(* PLC project waste_water_treatment_facility, Generated TextualNotationConverter 1.0 *)
(* stored: creationDateTime 2025-07-30T12:00:00, modificationDateTime 2025-01-30T12:00:00 *)

FUNCTION_BLOCK ANALOG_IN
  VAR_INPUT
    Name : STRING;
    Description : STRING;
    Raw_Signal : REAL;
    PV_High : REAL;
    PV_Low : REAL;
    Scaling_Slope : REAL;
    Scaling_Offset : REAL;
    Alarm_Enable : BOOL;
  END_VAR
  VAR_OUTPUT
    PV : REAL;
    High_Alarm : BOOL;
    Low_Alarm : BOOL;
    General_Fault : BOOL;
  END_VAR

            
          
END_FUNCTION_BLOCK

FUNCTION_BLOCK MOTOR_VSD
  VAR_INPUT
    Name : STRING;
    Description : STRING;
    Start_Cmd : BOOL;
    Stop_Cmd : BOOL;
    Speed_SP : REAL;
    Accel_Ramp : STRING;
    Decel_Ramp : STRING;
    Inhibit : BOOL;
  END_VAR
  VAR_OUTPUT
    Speed_Out : REAL;
    FB_Running : BOOL;
    FB_Fault : BOOL;
    FB_Ready : BOOL;
    FB_ActualSpeed : REAL;
    Alarm_Speed_Deviation : BOOL;
    Alarm_Comm_Fail : BOOL;
  END_VAR

            
          
END_FUNCTION_BLOCK

FUNCTION_BLOCK PID_BASIC
  VAR_INPUT
    Name : STRING;
    Description : STRING;
    AUTO : BOOL;
    PV : REAL;
    SP : REAL;
    MV_MIN : REAL;
    MV_MAX : REAL;
    X0 : REAL;
    KP : REAL;
    TR : REAL;
    TD : REAL;
    PV_High : REAL;
    PV_Low : REAL;
    Deviation_Limit : REAL;
    Inhibit : BOOL;
  END_VAR
  VAR_OUTPUT
    PV_High_Alarm : BOOL;
    PV_Low_Alarm : BOOL;
    Deviation_Alarm : BOOL;
    XOUT : REAL;
  END_VAR

            
          
END_FUNCTION_BLOCK

PROGRAM Section5
  VAR
    PH_401_pH_PV : REAL;
    AC_401_Alkalinity_PV : REAL;
    FT_101_InfluentFlow_PV : REAL;
    LT_401_TankLevel_PV : REAL;
    TS_401_Temperature_PV : REAL;
    PIC_401_pH_MV_Percent : REAL;
    PIC_402_Alkalinity_MV_Percent : REAL;
  END_VAR
  VAR
    AC-401 : ANALOG_IN;
    CD-401 : MOTOR_VSD;
    FT-101 : ANALOG_IN;
    LT-401 : ANALOG_IN;
    PH-401 : ANALOG_IN;
    PIC-401 : PID_BASIC;
    PIC-402 : PID_BASIC;
    TS-401 : ANALOG_IN;
  END_VAR
  VAR  (* added by the conversion: wires and edge detectors of the diagram *)
    _OR3_OUT : BOOL;
  END_VAR

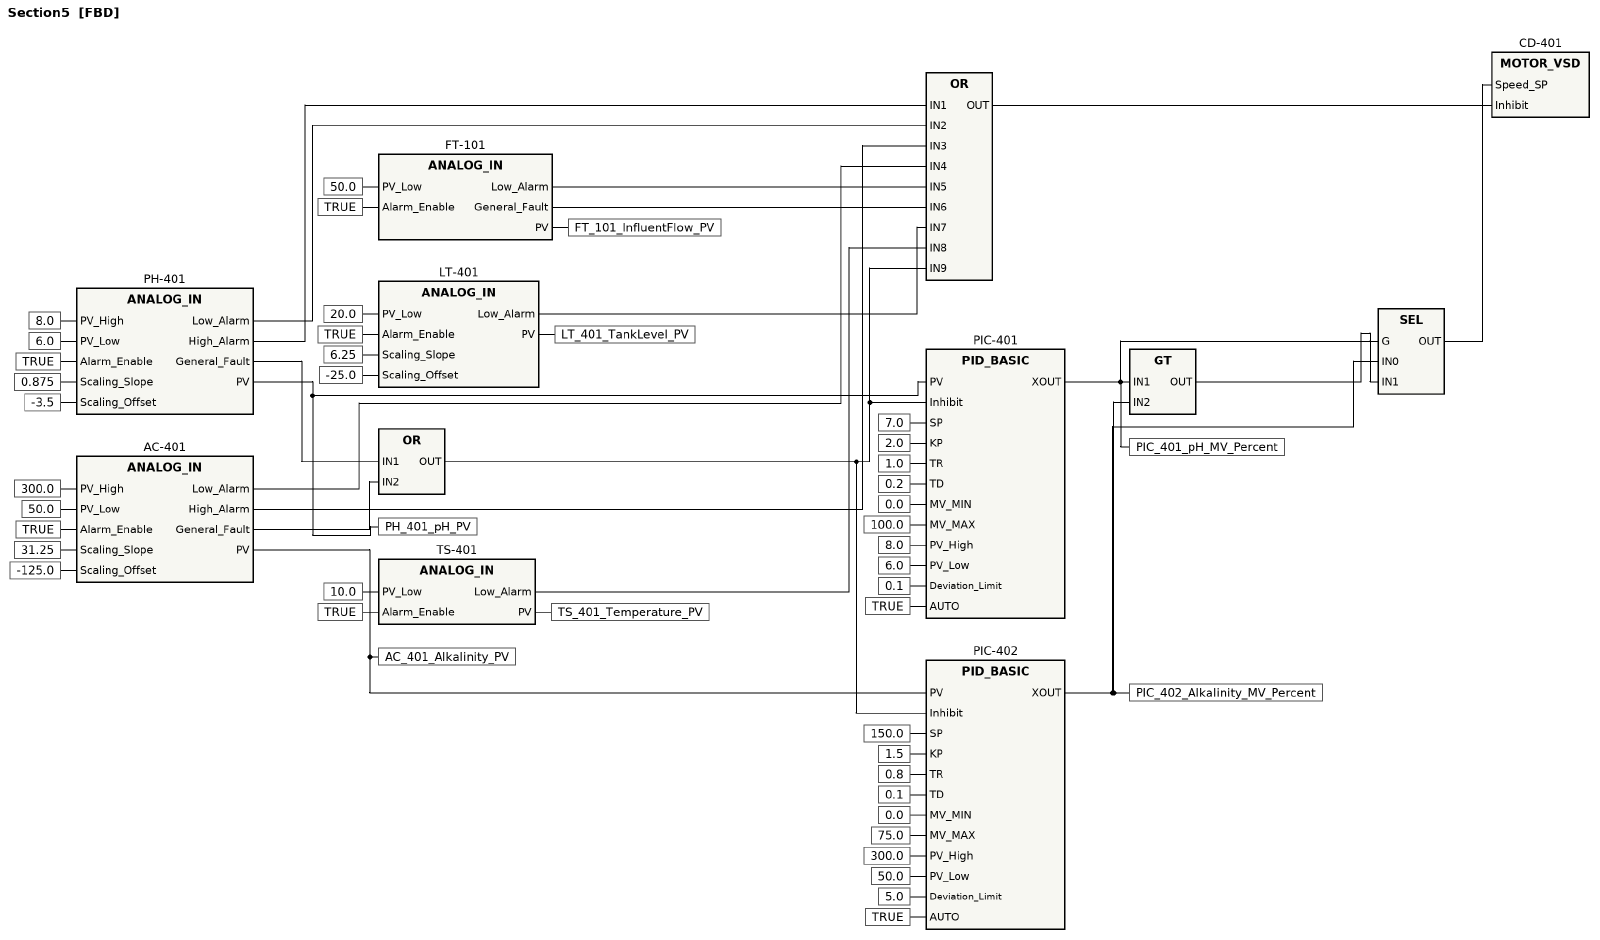
(* FBD diagram, written out as Structured Text *)
AC-401(PV_High := 300.0, PV_Low := 50.0, Alarm_Enable := TRUE, Scaling_Slope := 31.25, Scaling_Offset := -125.0);
AC_401_Alkalinity_PV := AC-401.PV;
FT-101(PV_Low := 50.0, Alarm_Enable := TRUE);
FT_101_InfluentFlow_PV := FT-101.PV;
LT-401(PV_Low := 20.0, Alarm_Enable := TRUE, Scaling_Slope := 6.25, Scaling_Offset := -25.0);
LT_401_TankLevel_PV := LT-401.PV;
PH-401(PV_High := 8.0, PV_Low := 6.0, Alarm_Enable := TRUE, Scaling_Slope := 0.875, Scaling_Offset := -3.5);
PH_401_pH_PV := PH-401.PV;
_OR3_OUT := PH-401.General_Fault OR AC-401.General_Fault;
PIC-401(PV := PH-401.PV, Inhibit := _OR3_OUT, SP := 7.0, KP := 2.0, TR := 1.0, TD := 0.2, MV_MIN := 0.0, MV_MAX := 100.0, PV_High := 8.0, PV_Low := 6.0, Deviation_Limit := 0.1, AUTO := TRUE);
PIC_401_pH_MV_Percent := PIC-401.XOUT;
PIC-402(PV := AC-401.PV, Inhibit := _OR3_OUT, SP := 150.0, KP := 1.5, TR := 0.8, TD := 0.1, MV_MIN := 0.0, MV_MAX := 75.0, PV_High := 300.0, PV_Low := 50.0, Deviation_Limit := 5.0, AUTO := TRUE);
PIC_402_Alkalinity_MV_Percent := PIC-402.XOUT;
TS-401(PV_Low := 10.0, Alarm_Enable := TRUE);
TS_401_Temperature_PV := TS-401.PV;
CD-401(Speed_SP := SEL(PIC-401.XOUT > PIC-402.XOUT, PIC-402.XOUT, PIC-401.XOUT), Inhibit := PH-401.High_Alarm OR PH-401.Low_Alarm OR AC-401.High_Alarm OR AC-401.Low_Alarm OR FT-101.Low_Alarm OR FT-101.General_Fault OR LT-401.Low_Alarm OR TS-401.Low_Alarm OR _OR3_OUT);
END_PROGRAM

FUNCTION_BLOCK BOOL_IN
  VAR_INPUT
    Name : STRING;
    Description : STRING;
    Bool_In : BOOL;
    Alarm_OnTrue : BOOL;
    Alarm_OnFalse : BOOL;
    Latch_Enable : BOOL;
    Reset_Latch : BOOL;
  END_VAR
  VAR_OUTPUT
    Bool_Out : BOOL;
    Alarm_Active : BOOL;
    Latched_Status : BOOL;
  END_VAR

            
          
END_FUNCTION_BLOCK

FUNCTION_BLOCK DIGITAL_IN
  VAR_INPUT
    Name : STRING;
    Description : STRING;
    DI_Raw : BOOL;
    DebounceTime : STRING;
    EnableAlarm : BOOL;
  END_VAR
  VAR_OUTPUT
    DI_Out : BOOL;
    Fault_State : BOOL;
  END_VAR

            
          
END_FUNCTION_BLOCK

FUNCTION_BLOCK DUTY_STANDBY
  VAR_INPUT
    Name : STRING;
    Description : STRING;
    Enable : BOOL;
    StartRequest : BOOL;
    AlternateEnable : BOOL;
    ForcePumpA : BOOL;
    ForcePumpB : BOOL;
    DutyElapsed : BOOL;
    MinRunElapsed : BOOL;
    SwitchoverDelayElapsed : BOOL;
    StartTimeoutElapsed : BOOL;
    PumpA_RunFB : BOOL;
    PumpB_RunFB : BOOL;
    PumpA_Fault : BOOL;
    PumpB_Fault : BOOL;
    Reset : BOOL;
    Inhibit : BOOL;
  END_VAR
  VAR_OUTPUT
    CmdPumpA : BOOL;
    CmdPumpB : BOOL;
    ActiveIsA : BOOL;
    SwitchedDueToDuty : BOOL;
    SwitchedDueToFailure : BOOL;
    Alarm_FailedStart_A : BOOL;
    Alarm_FailedStart_B : BOOL;
    Alarm_NoAvailablePump : BOOL;
  END_VAR

            
          
END_FUNCTION_BLOCK

FUNCTION_BLOCK MOTOR_2SPD
  VAR_INPUT
    Name : STRING;
    Description : STRING;
    Start_Cmd : BOOL;
    Stop_Cmd : BOOL;
    Speed_High_Cmd : BOOL;
    Speed_Low_Cmd : BOOL;
    Inhibit : BOOL;
  END_VAR
  VAR_OUTPUT
    Motor_Start_Out : BOOL;
    FB_Running : BOOL;
    FB_Trip : BOOL;
    FB_HighSpeed : BOOL;
    FB_LowSpeed : BOOL;
    Alarm_Speed_Error : BOOL;
  END_VAR

            
          
END_FUNCTION_BLOCK

FUNCTION_BLOCK MOTOR_ON_OFF
  VAR_INPUT
    Name : STRING;
    Description : STRING;
    Start_Cmd : BOOL;
    Stop_Cmd : BOOL;
    Start_Delay : STRING;
    MinRunTime : STRING;
    Inhibit : BOOL;
  END_VAR
  VAR_OUTPUT
    Motor_Start_Out : BOOL;
    FB_Running : BOOL;
    FB_Trip : BOOL;
    Alarm_Start_Fail : BOOL;
    Alarm_Stop_Fail : BOOL;
  END_VAR

            
          
END_FUNCTION_BLOCK

FUNCTION_BLOCK RATIO_CONTROL
  VAR_INPUT
    Name : STRING;
    Description : STRING;
    Auto : BOOL;
    PrimaryPV : REAL;
    SecondaryPV : REAL;
    RatioSP : REAL;
    Bias : REAL;
    TrimKp : REAL;
    TrimTi : STRING;
    MV_MIN : REAL;
    MV_MAX : REAL;
    ManOut : REAL;
    Inhibit : BOOL;
  END_VAR
  VAR_OUTPUT
    SlaveSP : REAL;
    ActiveRatio : REAL;
    RatioErr : REAL;
  END_VAR

            
          
END_FUNCTION_BLOCK

FUNCTION_BLOCK SPLIT_RANGE
  VAR_INPUT
    Name : STRING;
    Description : STRING;
    IN : REAL;
    Split_Point : REAL;
    Output1_Start : REAL;
    Output1_End : REAL;
    Output2_Start : REAL;
    Output2_End : REAL;
  END_VAR
  VAR_OUTPUT
    OUT1 : REAL;
    OUT2 : REAL;
  END_VAR

            
          
END_FUNCTION_BLOCK

FUNCTION_BLOCK VALVE_ELECTRIC
  VAR_INPUT
    Name : STRING;
    Description : STRING;
    Control_Signal : REAL;
    Manual_Mode : BOOL;
    Manual_Position : REAL;
    Open_Limit : REAL;
    Close_Limit : REAL;
    Timeout : STRING;
    Inhibit : BOOL;
  END_VAR
  VAR_OUTPUT
    Valve_Position : REAL;
    Feedback_Pos : REAL;
    Valve_Moving : BOOL;
    Position_Error : BOOL;
    Alarm : BOOL;
  END_VAR

            
          
END_FUNCTION_BLOCK

FUNCTION_BLOCK VALVE_ON_OFF
  VAR_INPUT
    Name : STRING;
    Description : STRING;
    Open_Cmd : BOOL;
    Close_Cmd : BOOL;
    Timeout : STRING;
    Inhibit : BOOL;
  END_VAR
  VAR_OUTPUT
    FB_Opened : BOOL;
    FB_Closed : BOOL;
    Valve_Open_Out : BOOL;
    Valve_Close_Out : BOOL;
    Alarm_Position_Error : BOOL;
    Alarm_General : BOOL;
  END_VAR

            
          
END_FUNCTION_BLOCK

FUNCTION_BLOCK VOTING_ANALOG
  VAR_INPUT
    Name : STRING;
    Description : STRING;
    Input1 : REAL;
    Input2 : REAL;
    Input3 : REAL;
    Deviation_Limit : REAL;
    Voting_Scheme : STRING;
    EnableAlarm : BOOL;
    Inhibit : BOOL;
  END_VAR
  VAR_OUTPUT
    Voted_Output : REAL;
    Sensor1_Fault : BOOL;
    Sensor2_Fault : BOOL;
    Sensor3_Fault : BOOL;
    Alarm_Voting_Error : BOOL;
    Healthy_Sensors_Count : INT;
  END_VAR

            
          
END_FUNCTION_BLOCK

PROGRAM Section6
  VAR
    FFIC-102_AirflowSP_for_FIC-103 : REAL;
    PT-501_AirHeaderPressure_PV : REAL;
    B-501A_Running_FB : BOOL;
    B-501B_Running_FB : BOOL;
    MX-501_Running_FB : BOOL;
    XV-105_Open_FB : BOOL;
    AirflowDeviationAlarm : BOOL;
    LowFlowAlarm : BOOL;
  END_VAR
  VAR
    B-501A : MOTOR_ON_OFF;
    B-501B : MOTOR_ON_OFF;
    FFIC-102 : RATIO_CONTROL;
    FIC-101 : PID_BASIC;
    FIC-103 : PID_BASIC;
    FV-102 : VALVE_ELECTRIC;
    MX-501 : MOTOR_ON_OFF;
    PT-501 : ANALOG_IN;
    XV-105 : VALVE_ON_OFF;
  END_VAR
  VAR  (* added by the conversion: wires and edge detectors of the diagram *)
    _OR61_IN4 : ANY;
    _OR61_IN3 : ANY;
    _OR61_IN5 : ANY;
    _OR61_IN6 : ANY;
    _OR61_IN1 : ANY;
    _OR61_IN2 : ANY;
    _OR61_OUT : ANY;
    _OR61_OUT_2 : BOOL;
    _OR63_IN2 : ANY;
    _OR63_OUT : ANY;
    _OR63_OUT_2 : BOOL;
    _OR58_IN2 : ANY;
    _OR58_OUT : BOOL;
  END_VAR

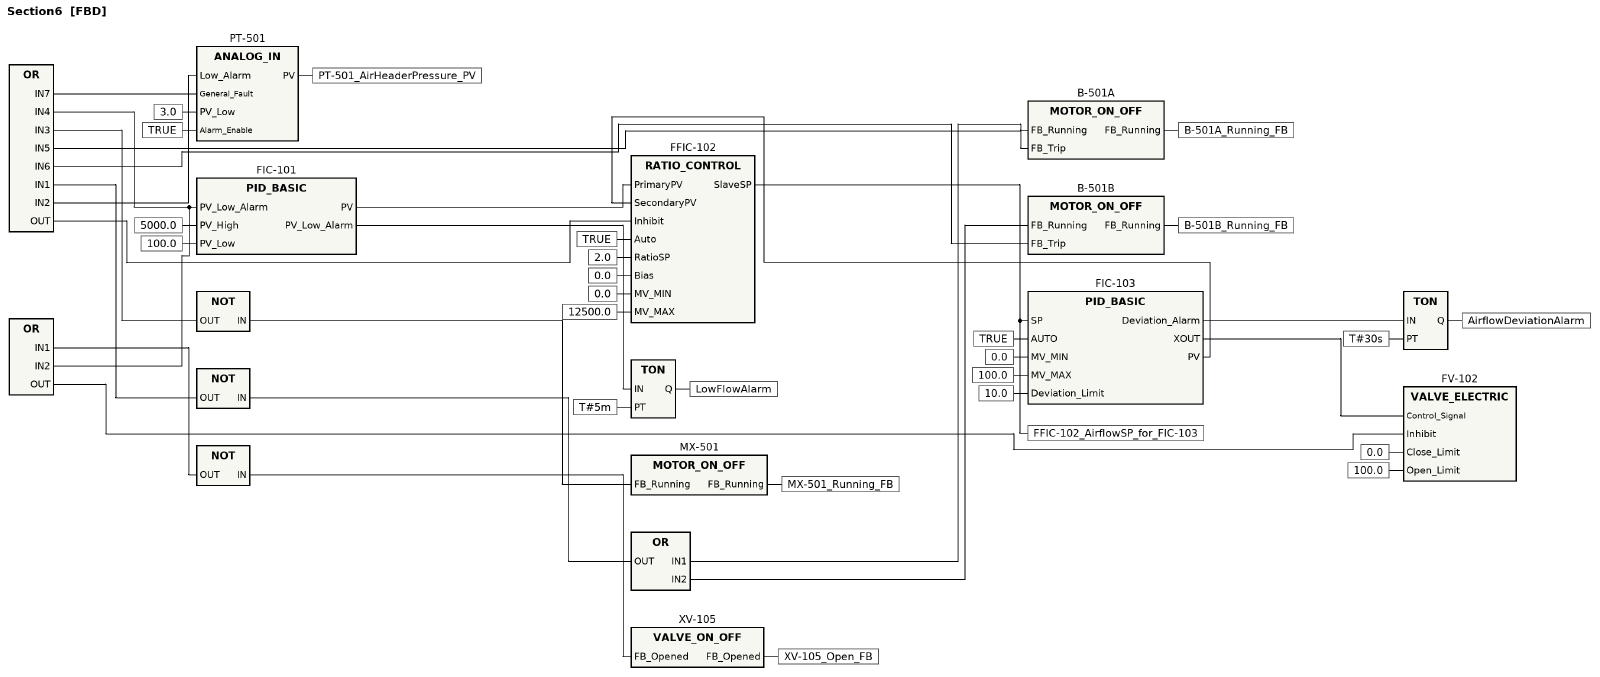
(* FBD diagram, written out as Structured Text *)
_OR61_OUT_2 := OR(IN4 => _OR61_IN4, IN3 => _OR61_IN3, IN5 => _OR61_IN5, IN6 => _OR61_IN6, IN1 => _OR61_IN1, IN2 => _OR61_IN2, OUT => _OR61_OUT);
_OR63_OUT_2 := OR(IN2 => _OR63_IN2, OUT => _OR63_OUT);
FIC-101(PV_Low_Alarm := _OR61_IN4 OR _OR63_IN2, PV_High := 5000.0, PV_Low := 100.0);
FFIC-102(PrimaryPV := FIC-101.PV, SecondaryPV := FIC-103.PV, Inhibit := _OR61_OUT, Auto := TRUE, RatioSP := 2.0, Bias := 0.0, MV_MIN := 0.0, MV_MAX := 12500.0);
FIC-103(SP := FFIC-102.SlaveSP, AUTO := TRUE, MV_MIN := 0.0, MV_MAX := 100.0, Deviation_Limit := 10.0);
AirflowDeviationAlarm := TON(FIC-103.Deviation_Alarm, T#30s);
_OR58_OUT := OR(OUT := NOT _OR61_IN1, IN2 => _OR58_IN2);
B-501A(FB_Running := _OR58_OUT, FB_Trip := _OR61_IN5);
B-501A_Running_FB := B-501A.FB_Running;
B-501B(FB_Running := _OR58_IN2, FB_Trip := _OR61_IN6);
B-501B_Running_FB := B-501B.FB_Running;
FFIC-102_AirflowSP_for_FIC-103 := FFIC-102.SlaveSP;
LowFlowAlarm := TON(FIC-101.PV_Low_Alarm, T#5m);
MX-501(FB_Running := NOT _OR61_IN3);
MX-501_Running_FB := MX-501.FB_Running;
PT-501(Low_Alarm := _OR61_IN2, General_Fault := _OR61_OUT_2, PV_Low := 3.0, Alarm_Enable := TRUE);
PT-501_AirHeaderPressure_PV := PT-501.PV;
XV-105(FB_Opened := NOT _OR63_OUT_2);
XV-105_Open_FB := XV-105.FB_Opened;
FV-102(Control_Signal := FIC-103.XOUT, Inhibit := _OR63_OUT, Close_Limit := 0.0, Open_Limit := 100.0);
END_PROGRAM

PROGRAM Section7
  VAR
    PT_601A_DischargePressure_PV : REAL;
    PT_601B_DischargePressure_PV : REAL;
    LS_601_BlanketLevelSwitchStatus : BOOL;
    CL_601A_Running : BOOL;
    CL_601B_Running : BOOL;
    PS_601A_Running : BOOL;
    PS_601B_Running : BOOL;
    VS_601A_Feedback_Position_Pct : REAL;
    VS_601B_Feedback_Position_Pct : REAL;
    CL_601_ActiveIsA : BOOL;
    PS_601_ActiveIsA : BOOL;
    CL_601A_RunCmd : BOOL;
    CL_601B_RunCmd : BOOL;
    PS_601A_RunCmd : BOOL;
    PS_601B_RunCmd : BOOL;
  END_VAR
  VAR
    LS-601 : BOOL_IN;
    PT-601A : ANALOG_IN;
    PT-601B : ANALOG_IN;
    CL-601A : MOTOR_ON_OFF;
    CL-601B : MOTOR_ON_OFF;
    PS-601A : MOTOR_ON_OFF;
    PS-601B : MOTOR_ON_OFF;
    VS-601A : VALVE_ELECTRIC;
    VS-601B : VALVE_ELECTRIC;
    CL-601_DUTY_STANDBY : DUTY_STANDBY;
    PS-601_DUTY_STANDBY : DUTY_STANDBY;
  END_VAR
  VAR  (* added by the conversion: wires and edge detectors of the diagram *)
    _OR110_OUT : BOOL;
    _OR113_OUT : BOOL;
    _OR114_OUT : BOOL;
    _OR100_OUT : BOOL;
    _OR115_OUT : BOOL;
    _OR105_OUT : BOOL;
  END_VAR

(* FBD diagram, written out as Structured Text *)
LS-601(Alarm_OnTrue := TRUE, Alarm_OnFalse := FALSE, Latch_Enable := TRUE);
_OR110_OUT := LS-601.Bool_Out OR LS-601.Alarm_Active;
_OR113_OUT := _OR110_OUT OR CL-601A.FB_Trip;
CL-601A(Start_Cmd := CL-601_DUTY_STANDBY.CmdPumpA, Inhibit := _OR113_OUT, Start_Delay := T#5S, MinRunTime := T#30M);
_OR114_OUT := _OR110_OUT OR CL-601B.FB_Trip;
CL-601B(Start_Cmd := CL-601_DUTY_STANDBY.CmdPumpB, Inhibit := _OR114_OUT, Start_Delay := T#5S, MinRunTime := T#30M);
_OR100_OUT := CL-601A.FB_Running OR CL-601B.FB_Running;
PT-601A(PV_Low := 25.0, Alarm_Enable := TRUE);
PT-601B(PV_Low := 25.0, Alarm_Enable := TRUE);
_OR115_OUT := _OR110_OUT OR PT-601A.Low_Alarm OR PT-601B.Low_Alarm;
CL-601_DUTY_STANDBY(DutyElapsed := TON(_OR100_OUT, T#72H), MinRunElapsed := TON(_OR100_OUT, T#30M), SwitchoverDelayElapsed := TON(NOT _OR100_OUT, T#10S), PumpA_RunFB := CL-601A.FB_Running, PumpB_RunFB := CL-601B.FB_Running, PumpA_Fault := _OR113_OUT, PumpB_Fault := _OR114_OUT, Inhibit := _OR115_OUT, Enable := TRUE, StartRequest := TRUE, AlternateEnable := TRUE);
CL_601A_RunCmd := CL-601_DUTY_STANDBY.CmdPumpA;
CL_601A_Running := CL-601A.FB_Running;
CL_601B_RunCmd := CL-601_DUTY_STANDBY.CmdPumpB;
CL_601B_Running := CL-601B.FB_Running;
CL_601_ActiveIsA := CL-601_DUTY_STANDBY.ActiveIsA;
LS_601_BlanketLevelSwitchStatus := LS-601.Bool_Out;
PS-601A(Start_Cmd := PS-601_DUTY_STANDBY.CmdPumpA, Inhibit := PT-601A.Low_Alarm OR _OR110_OUT, Start_Delay := T#5S, MinRunTime := T#30M);
PS-601B(Start_Cmd := PS-601_DUTY_STANDBY.CmdPumpB, Inhibit := PT-601B.Low_Alarm OR _OR110_OUT, Start_Delay := T#5S, MinRunTime := T#30M);
_OR105_OUT := PS-601A.FB_Running OR PS-601B.FB_Running;
PS-601_DUTY_STANDBY(DutyElapsed := TON(_OR105_OUT, T#72H), MinRunElapsed := TON(_OR105_OUT, T#30M), SwitchoverDelayElapsed := TON(NOT _OR105_OUT, T#10S), PumpA_RunFB := PS-601A.FB_Running, PumpB_RunFB := PS-601B.FB_Running, Inhibit := _OR115_OUT, PumpA_Fault := PS-601A.FB_Trip OR PT-601A.Low_Alarm, PumpB_Fault := PS-601B.FB_Trip OR PT-601B.Low_Alarm, Enable := TRUE, StartRequest := TRUE, AlternateEnable := TRUE);
PS_601A_RunCmd := PS-601_DUTY_STANDBY.CmdPumpA;
PS_601A_Running := PS-601A.FB_Running;
PS_601B_RunCmd := PS-601_DUTY_STANDBY.CmdPumpB;
PS_601B_Running := PS-601B.FB_Running;
PS_601_ActiveIsA := PS-601_DUTY_STANDBY.ActiveIsA;
PT_601A_DischargePressure_PV := PT-601A.PV;
PT_601B_DischargePressure_PV := PT-601B.PV;
VS-601A(Open_Limit := 100.0, Close_Limit := 0.0);
VS_601A_Feedback_Position_Pct := VS-601A.Feedback_Pos;
VS-601B(Open_Limit := 100.0, Close_Limit := 0.0);
VS_601B_Feedback_Position_Pct := VS-601B.Feedback_Pos;
END_PROGRAM

PROGRAM Section8
  VAR
    FT701_InfluentFlow_PV : REAL;
    FT702_BackwashFlow_PV : REAL;
    FIC702_BackwashFlow_SP : REAL;
    FFIC703_ActiveRatio : REAL;
    TT701_Turbidity_PV : REAL;
    TF701_InOperation : BOOL;
  END_VAR
  VAR
    FFIC-703 : RATIO_CONTROL;
    FIC-702 : PID_BASIC;
    FT-701 : ANALOG_IN;
    FT-702 : ANALOG_IN;
    FV-702 : VALVE_ELECTRIC;
    TT-701 : ANALOG_IN;
    TF-701 : BOOL_IN;
  END_VAR
  VAR  (* added by the conversion: wires and edge detectors of the diagram *)
    _OR175_OUT : BOOL;
  END_VAR

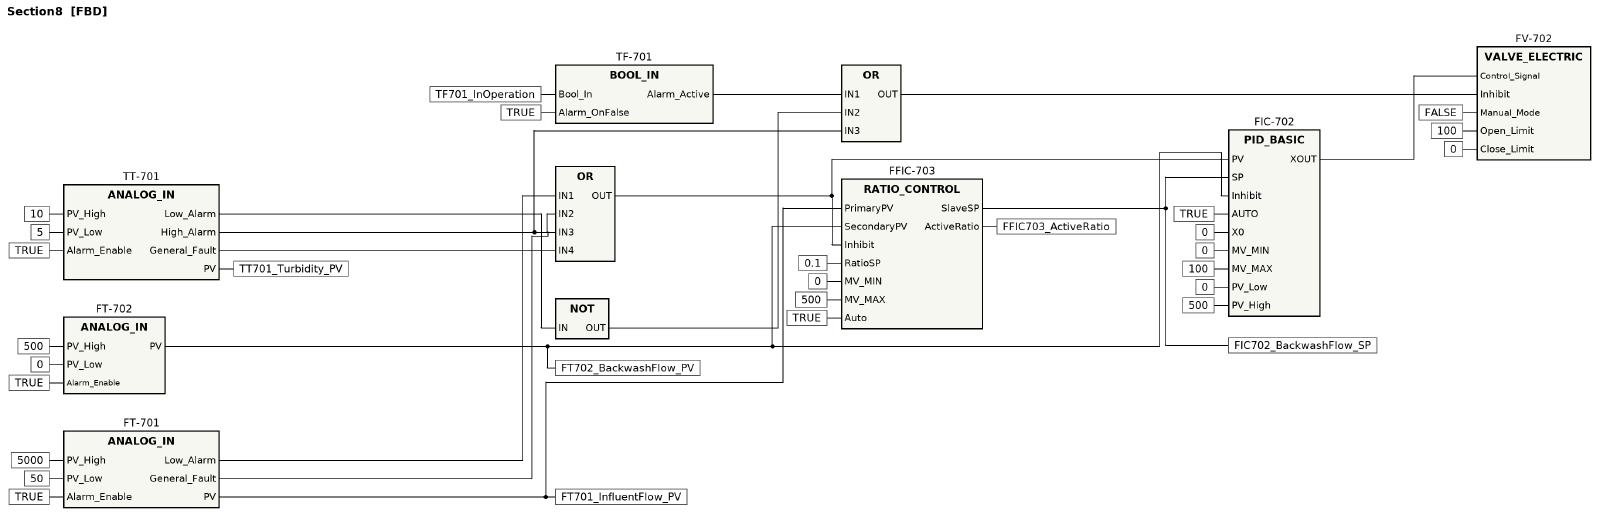
(* FBD diagram, written out as Structured Text *)
FT-701(PV_High := 5000, PV_Low := 50, Alarm_Enable := TRUE);
FT-702(PV_High := 500, PV_Low := 0, Alarm_Enable := TRUE);
TT-701(PV_High := 10, PV_Low := 5, Alarm_Enable := TRUE);
_OR175_OUT := FT-701.Low_Alarm OR TT-701.High_Alarm OR FT-701.General_Fault OR TT-701.General_Fault;
FFIC-703(PrimaryPV := FT-701.PV, SecondaryPV := FT-702.PV, Inhibit := _OR175_OUT, RatioSP := 0.1, MV_MIN := 0, MV_MAX := 500, Auto := TRUE);
FFIC703_ActiveRatio := FFIC-703.ActiveRatio;
FIC702_BackwashFlow_SP := FFIC-703.SlaveSP;
FT701_InfluentFlow_PV := FT-701.PV;
FT702_BackwashFlow_PV := FT-702.PV;
TT701_Turbidity_PV := TT-701.PV;
TF-701(Bool_In := TF701_InOperation, Alarm_OnFalse := TRUE);
FIC-702(PV := FT-702.PV, SP := FFIC-703.SlaveSP, Inhibit := _OR175_OUT, AUTO := TRUE, X0 := 0, MV_MIN := 0, MV_MAX := 100, PV_Low := 0, PV_High := 500);
FV-702(Control_Signal := FIC-702.XOUT, Inhibit := TF-701.Alarm_Active OR NOT TT-701.Low_Alarm OR TT-701.High_Alarm, Manual_Mode := FALSE, Open_Limit := 100, Close_Limit := 0);
END_PROGRAM

PROGRAM Section9
  VAR
    FT801_EffluentFlow_PV_m3h : REAL;
    FTCL801_ChlorineFlow_PV_m3h : REAL;
    FTDC801_DechlorFlow_PV_m3h : REAL;
    CL801_DoseFlow_SP_m3h : REAL;
    DC801_DoseFlow_SP_m3h : REAL;
  END_VAR
  VAR
    FT-801 : ANALOG_IN;
    FT-CL-801 : ANALOG_IN;
    FT-DC-801 : ANALOG_IN;
    FIC-101 : RATIO_CONTROL;
    FIC-102 : RATIO_CONTROL;
    LV-105 : VALVE_ELECTRIC;
    XV-106 : VALVE_ON_OFF;
    XV-106-OPEN-LS : DIGITAL_IN;
    XV-106-CLOSED-LS : DIGITAL_IN;
    CL-801 : MOTOR_VSD;
    DC-801 : MOTOR_VSD;
    UV-801 : MOTOR_ON_OFF;
  END_VAR
  VAR  (* added by the conversion: wires and edge detectors of the diagram *)
    _OR218_OUT : BOOL;
  END_VAR

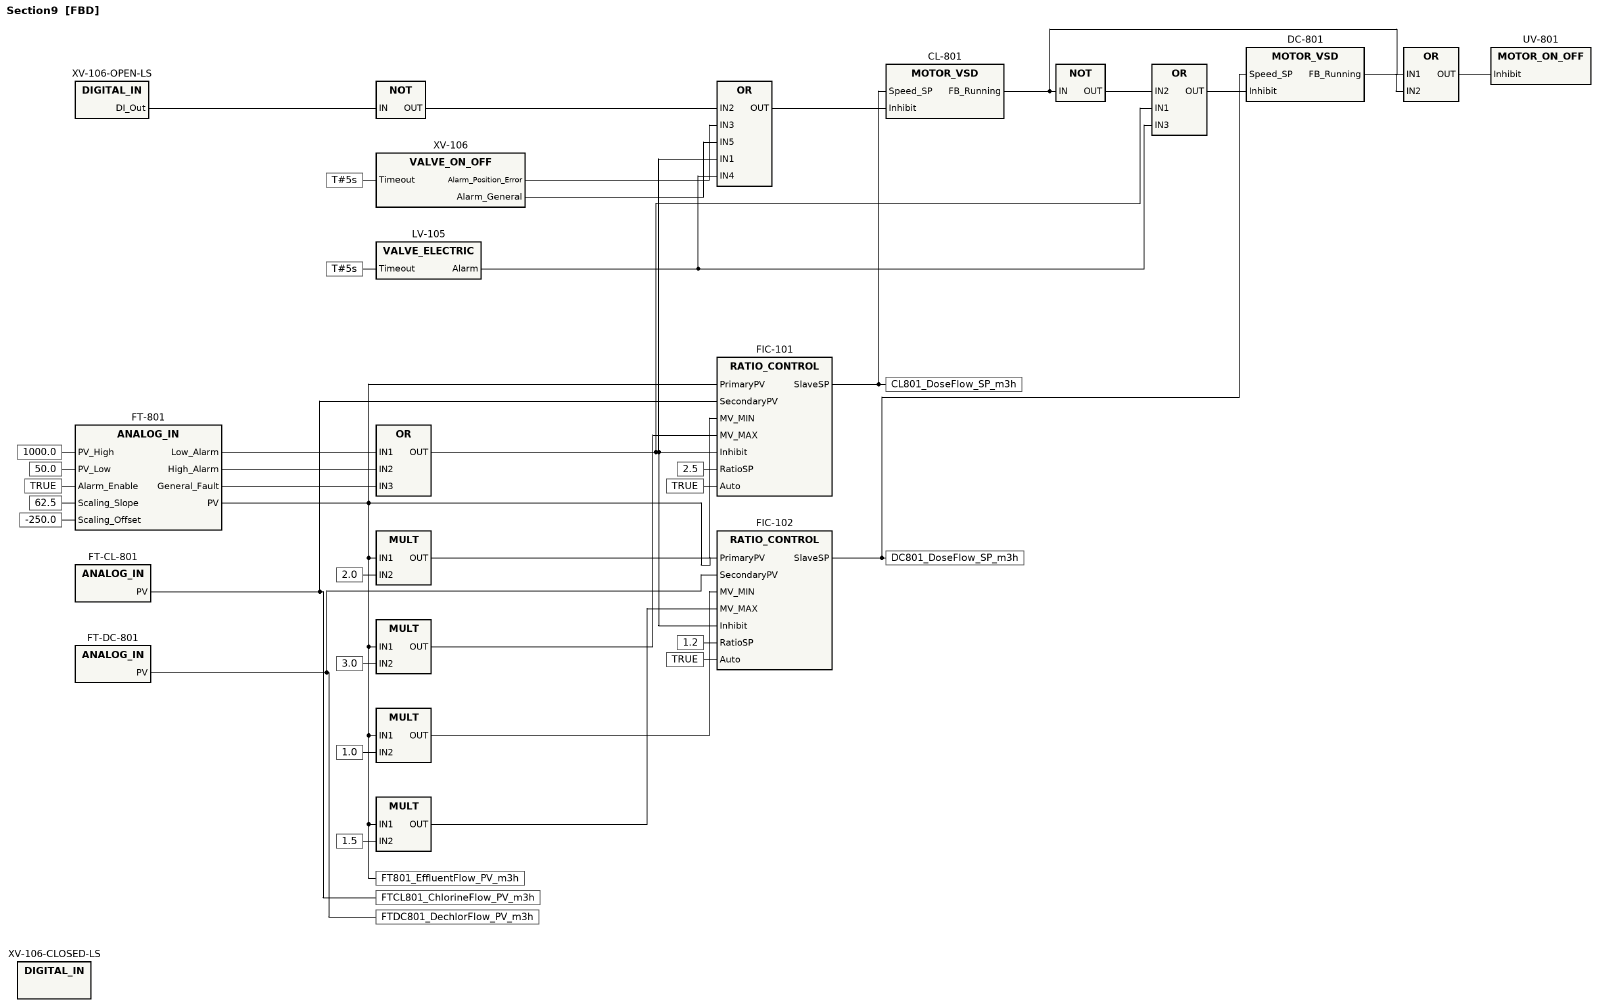
(* FBD diagram, written out as Structured Text *)
FT-801(PV_High := 1000.0, PV_Low := 50.0, Alarm_Enable := TRUE, Scaling_Slope := 62.5, Scaling_Offset := -250.0);
FT-CL-801();
_OR218_OUT := FT-801.Low_Alarm OR FT-801.High_Alarm OR FT-801.General_Fault;
FIC-101(PrimaryPV := FT-801.PV, SecondaryPV := FT-CL-801.PV, MV_MIN := MULT(FT-801.PV, 2.0), MV_MAX := MULT(FT-801.PV, 3.0), Inhibit := _OR218_OUT, RatioSP := 2.5, Auto := TRUE);
CL801_DoseFlow_SP_m3h := FIC-101.SlaveSP;
FT-DC-801();
FIC-102(PrimaryPV := FT-801.PV, SecondaryPV := FT-DC-801.PV, MV_MIN := MULT(FT-801.PV, 1.0), MV_MAX := MULT(FT-801.PV, 1.5), Inhibit := _OR218_OUT, RatioSP := 1.2, Auto := TRUE);
DC801_DoseFlow_SP_m3h := FIC-102.SlaveSP;
FT801_EffluentFlow_PV_m3h := FT-801.PV;
FTCL801_ChlorineFlow_PV_m3h := FT-CL-801.PV;
FTDC801_DechlorFlow_PV_m3h := FT-DC-801.PV;
XV-106-OPEN-LS();
XV-106(Timeout := T#5s);
LV-105(Timeout := T#5s);
CL-801(Speed_SP := FIC-101.SlaveSP, Inhibit := NOT XV-106-OPEN-LS.DI_Out OR XV-106.Alarm_Position_Error OR XV-106.Alarm_General OR _OR218_OUT OR LV-105.Alarm);
DC-801(Speed_SP := FIC-102.SlaveSP, Inhibit := NOT CL-801.FB_Running OR _OR218_OUT OR LV-105.Alarm);
XV-106-CLOSED-LS();
UV-801(Inhibit := CL-801.FB_Running OR DC-801.FB_Running);
END_PROGRAM

PROGRAM Section10
  VAR
    FT-901_Flow_PV : REAL;
    LS-901_Level_PV : REAL;
    P-901A_MotorStartOut : BOOL;
    P-901B_MotorStartOut : BOOL;
    XV-102_CloseOut : BOOL;
  END_VAR
  VAR
    FT-901 : ANALOG_IN;
    LS-901 : ANALOG_IN;
    P-901A : MOTOR_ON_OFF;
    P-901B : MOTOR_ON_OFF;
    XV-102 : VALVE_ON_OFF;
    P-901_DS : DUTY_STANDBY;
  END_VAR
  VAR  (* added by the conversion: wires and edge detectors of the diagram *)
    _GT258_OUT : BOOL;
    _OR274_OUT : BOOL;
    _AND268_OUT : BOOL;
    _OR263_OUT : BOOL;
    _AND266_OUT : BOOL;
    _TON267_OUT : BOOL;
    _TON269_OUT : BOOL;
    _OR272_OUT : BOOL;
  END_VAR

(* FBD diagram, written out as Structured Text *)
FT-901(PV_Low := 15.0, Alarm_Enable := TRUE);
FT-901_Flow_PV := FT-901.PV;
LS-901(PV_Low := 40.0, PV_High := 90.0, Alarm_Enable := TRUE);
LS-901_Level_PV := LS-901.PV;
_GT258_OUT := LS-901.PV > 85.0;
_OR274_OUT := P-901_DS.CmdPumpB OR _GT258_OUT;
_AND268_OUT := P-901B.FB_Running AND FT-901.Low_Alarm;
P-901B(Start_Cmd := _OR274_OUT, Stop_Cmd := NOT _OR274_OUT, Inhibit := LS-901.Low_Alarm OR _AND268_OUT, MinRunTime := T#30m);
_OR263_OUT := P-901_DS.ActiveIsA AND P-901A.FB_Running OR NOT P-901_DS.ActiveIsA AND P-901B.FB_Running;
_AND266_OUT := P-901A.FB_Running AND FT-901.Low_Alarm;
_TON267_OUT := TON(_AND266_OUT, T#10s);
_TON269_OUT := TON(_AND268_OUT, T#10s);
P-901_DS(DutyElapsed := TON(_OR263_OUT, T#48h), MinRunElapsed := TON(_OR263_OUT, T#30m), PumpA_Fault := _TON267_OUT, PumpB_Fault := _TON269_OUT, SwitchoverDelayElapsed := TON(_TON267_OUT OR _TON269_OUT, T#5s), StartRequest := RS(LS-901.PV > 60.0, LS-901.PV < 40.0), PumpA_RunFB := P-901A.FB_Running, PumpB_RunFB := P-901B.FB_Running, Enable := TRUE, AlternateEnable := TRUE);
_OR272_OUT := P-901_DS.CmdPumpA OR _GT258_OUT;
P-901A(Start_Cmd := _OR272_OUT, Stop_Cmd := NOT _OR272_OUT, Inhibit := LS-901.Low_Alarm OR _AND266_OUT, MinRunTime := T#30m);
P-901A_MotorStartOut := P-901A.Motor_Start_Out;
P-901B_MotorStartOut := P-901B.Motor_Start_Out;
XV-102(Inhibit := P-901_DS.Alarm_NoAvailablePump, Close_Cmd := P-901_DS.Alarm_NoAvailablePump);
XV-102_CloseOut := XV-102.Valve_Close_Out;
END_PROGRAM

PROGRAM Section11
  VAR
    FIT104_InfluentFlow_PV : REAL;
    FFIC107_ChemDose_SlaveSP : REAL;
    FFIC107_ActiveRatio : REAL;
  END_VAR
  VAR
    FIT-104 : ANALOG_IN;
    FFIC-107 : RATIO_CONTROL;
    FIC-106 : PID_BASIC;
    CD-1001 : MOTOR_VSD;
    PV-101 : VALVE_ELECTRIC;
    XV-102 : VALVE_ON_OFF;
  END_VAR

(* FBD diagram, written out as Structured Text *)
FIT-104(Name := "Influent Flow FIT-104", Scaling_Slope := 312.5, Scaling_Offset := -1250.0, PV_High := 5000.0, PV_Low := 100.0, Alarm_Enable := TRUE);
FIC-106(SP := FFIC-107.SlaveSP, PV := CD-1001.FB_ActualSpeed, Name := "Chemical Dosing PID FIC-106", AUTO := TRUE, MV_MIN := 0.0, MV_MAX := 100.0, X0 := 0.0, KP := 1.0, TR := 10.0, TD := 0.0, PV_High := 100.0, PV_Low := 0.0, Deviation_Limit := 3.0);
XV-102(Name := "Shut-off Valve XV-102", Timeout := T#5s);
PV-101(Name := "Pressure Control Valve PV-101", Open_Limit := 100.0, Close_Limit := 0.0, Timeout := T#5s);
CD-1001(Speed_SP := FIC-106.XOUT, Inhibit := NOT XV-102.FB_Opened OR PV-101.Alarm OR PV-101.Position_Error OR XV-102.Alarm_Position_Error OR XV-102.Alarm_General, Name := "Chemical Dosing Pump CD-1001", Accel_Ramp := T#2s, Decel_Ramp := T#2s);
FFIC-107(PrimaryPV := FIT-104.PV, SecondaryPV := CD-1001.FB_ActualSpeed, Inhibit := FIT-104.Low_Alarm OR FIT-104.General_Fault OR CD-1001.FB_Fault OR CD-1001.Alarm_Comm_Fail OR CD-1001.Alarm_Speed_Deviation, Name := "Chemical Ratio Controller FFIC-107", Auto := TRUE, RatioSP := 2.5, Bias := 0.0, TrimKp := 0.0, TrimTi := T#0s, MV_MIN := 0.0, MV_MAX := 15000.0);
FFIC107_ActiveRatio := FFIC-107.ActiveRatio;
FFIC107_ChemDose_SlaveSP := FFIC-107.SlaveSP;
FIT104_InfluentFlow_PV := FIT-104.PV;
END_PROGRAM

PROGRAM Section12
  VAR
    IIC101_Solids_PV : REAL;
    PV102_MV_Command : REAL;
    LV104_Level_PV : REAL;
  END_VAR
  VAR
    IIC-101 : ANALOG_IN;
    IIC-103 : PID_BASIC;
    LV-104 : ANALOG_IN;
    PV-102 : VALVE_ELECTRIC;
    OC-1101 : VALVE_ON_OFF;
    DG-1101 : BOOL_IN;
    DW-1101 : BOOL_IN;
    IIC-105 : BOOL_IN;
  END_VAR
  VAR  (* added by the conversion: wires and edge detectors of the diagram *)
    _OR353_OUT : BOOL;
  END_VAR

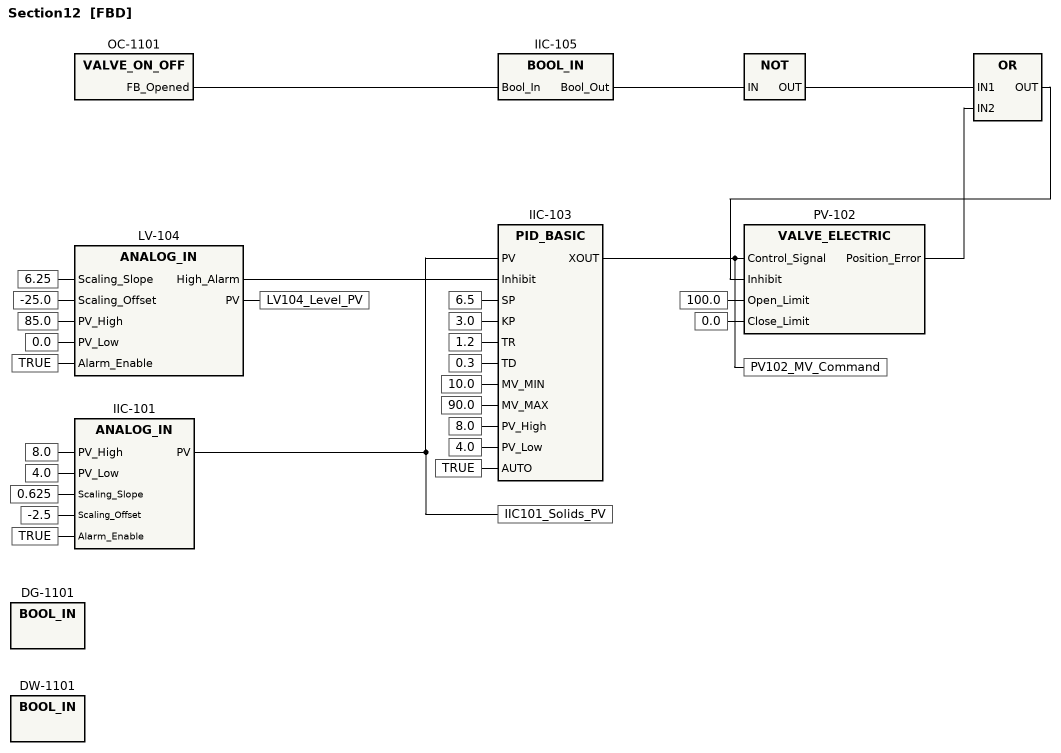
(* FBD diagram, written out as Structured Text *)
IIC-101(PV_High := 8.0, PV_Low := 4.0, Scaling_Slope := 0.625, Scaling_Offset := -2.5, Alarm_Enable := TRUE);
IIC101_Solids_PV := IIC-101.PV;
LV-104(Scaling_Slope := 6.25, Scaling_Offset := -25.0, PV_High := 85.0, PV_Low := 0.0, Alarm_Enable := TRUE);
LV104_Level_PV := LV-104.PV;
IIC-103(PV := IIC-101.PV, Inhibit := LV-104.High_Alarm, SP := 6.5, KP := 3.0, TR := 1.2, TD := 0.3, MV_MIN := 10.0, MV_MAX := 90.0, PV_High := 8.0, PV_Low := 4.0, AUTO := TRUE);
PV102_MV_Command := IIC-103.XOUT;
OC-1101();
IIC-105(Bool_In := OC-1101.FB_Opened);
PV-102(Control_Signal := IIC-103.XOUT, Inhibit := _OR353_OUT, Open_Limit := 100.0, Close_Limit := 0.0);
_OR353_OUT := NOT IIC-105.Bool_Out OR PV-102.Position_Error;
DG-1101();
DW-1101();
END_PROGRAM

CONFIGURATION Config0
  RESOURCE Res0 ON PLC
    TASK task0(INTERVAL := T#20ms, PRIORITY := 0);
    PROGRAM instance0 WITH task0 : Section5;
    PROGRAM instance_1 WITH task0 : Section6;
    PROGRAM instance_2 WITH task0 : Section7;
    PROGRAM instance_3 WITH task0 : Section8;
    PROGRAM instance_4 WITH task0 : Section9;
    PROGRAM instance_5 WITH task0 : Section10;
    PROGRAM instance_6 WITH task0 : Section11;
    PROGRAM instance_7 WITH task0 : Section12;
  END_RESOURCE
END_CONFIGURATION
